{attribute 'qualified_only'}
FUNCTION_BLOCK FB_ConveyorControl
VAR_INPUT
	// Control inputs
	bStart			: BOOL;		// Start conveyor command
	bReset			: BOOL;		// Reset faults and errors
	nSpeed			: INT;		// Desired speed percentage (0-100)
END_VAR
VAR_OUTPUT
	// Status outputs
	bRunning		: BOOL;		// Conveyor is running
	bFault			: BOOL;		// Fault condition present
	bReady			: BOOL;		// Ready to start
	nActualSpeed	: INT;		// Actual speed percentage
END_VAR
VAR
	// Internal variables
	eState			: E_MotorState;		// Current motor state
	stConveyorData	: ST_ConveyorData;	// Conveyor configuration data
	
	// Timers
	tonStartDelay	: TON;		// Start delay timer
	tonRunTime		: TON;		// Running time counter
	tonFaultDelay	: TON;		// Fault detection delay
	
	// Internal flags
	bInternalFault	: BOOL;		// Internal fault flag
	bStartRequest	: BOOL;		// Start request edge detection
	bLastStart		: BOOL;		// Previous start signal
	
	// Counters
	nStartCount		: UDINT;	// Number of starts
	nRunTimeHours	: UDINT;	// Running time in hours
END_VAR

// =====================================================
// FB_ConveyorControl - Conveyor Control Function Block
// Purpose: Control conveyor motor with safety features
// Author: Demo System  
// Version: 1.0
// =====================================================

// Edge detection for start command
bStartRequest := bStart AND NOT bLastStart;
bLastStart := bStart;

// Count start requests
IF bStartRequest THEN
	nStartCount := nStartCount + 1;
END_IF

// Reset logic
IF NOT bReset THEN
	bInternalFault := FALSE;
	eState := E_MotorState.STOPPED;
END_IF

// Main state machine
CASE eState OF
	E_MotorState.STOPPED:
		// Conveyor stopped state
		bRunning := FALSE;
		bReady := TRUE;
		nActualSpeed := 0;
		
		// Check for start condition
		IF bStart AND bReset AND NOT bInternalFault THEN
			eState := E_MotorState.STARTING;
			tonStartDelay(IN := TRUE, PT := T#2S);
		END_IF
		
	E_MotorState.STARTING:
		// Starting sequence
		bRunning := FALSE;
		bReady := FALSE;
		
		tonStartDelay(IN := TRUE);
		IF tonStartDelay.Q THEN
			eState := E_MotorState.RUNNING;
			tonStartDelay(IN := FALSE);
			tonRunTime(IN := TRUE);
		END_IF
		
		// Check for abort conditions
		IF NOT bStart OR NOT bReset THEN
			eState := E_MotorState.STOPPING;
		END_IF
		
	E_MotorState.RUNNING:
		// Normal running state
		bRunning := TRUE;
		bReady := FALSE;
		
		// Speed control (simplified)
		IF nSpeed > 100 THEN
			nActualSpeed := 100;
		ELSIF nSpeed < 0 THEN
			nActualSpeed := 0;
		ELSE
			nActualSpeed := nSpeed;
		END_IF
		
		// Running time counter
		tonRunTime(IN := TRUE);
		
		// Check for stop conditions
		IF NOT bStart OR NOT bReset OR bInternalFault THEN
			eState := E_MotorState.STOPPING;
		END_IF
		
	E_MotorState.STOPPING:
		// Stopping sequence
		bRunning := FALSE;
		bReady := FALSE;
		nActualSpeed := 0;
		
		tonRunTime(IN := FALSE);
		eState := E_MotorState.STOPPED;
		
	E_MotorState.FAULT:
		// Fault state
		bRunning := FALSE;
		bReady := FALSE;
		bFault := TRUE;
		nActualSpeed := 0;
		
		// Reset from fault
		IF bReset THEN
			eState := E_MotorState.STOPPED;
			bFault := FALSE;
		END_IF
		
	ELSE
		// Invalid state - go to fault
		eState := E_MotorState.FAULT;
		bInternalFault := TRUE;
END_CASE

// Fault detection logic
tonFaultDelay(IN := (nActualSpeed > 95 AND bRunning), PT := T#30S);
IF tonFaultDelay.Q THEN
	bInternalFault := TRUE;
	eState := E_MotorState.FAULT;
END_IF

// Update conveyor data structure
stConveyorData.bRunning := bRunning;
stConveyorData.nSpeed := nActualSpeed;
stConveyorData.nStartCount := nStartCount;
stConveyorData.tRunTime := UDINT_TO_TIME(tonRunTime.ET);

END_FUNCTION_BLOCK

(* stored: Version 1.1.0.1, ProductVersion 3.5.13.50
   POU FB_ConveyorControl: Id {3dc6b881-9d15-491e-8f3c-929d5ca9c872}, SpecialFunc None *)
